Yaskawa INFORM job: UF_SELECTIE.JBI

/JOB
//NAME UF_SELECTIE
//POS
///NPOS 0,0,0,6,0,0
///USER 15
///TOOL 1
///POSTYPE USER
///RECTAN
///RCONF 1,0,0,0,0,0,0,0,0,0,0,0,0,0,0,0,0,0,0,0,0,0,0,0
P00100=0.001,-0.002,0.001,159.0512,-20.0126,15.9786
///USER 16
///RCONF 0,0,0,0,1,0,0,0,0,0,0,0,0,0,0,0,0,0,0,0,0,0,0,0
P00101=0.509,-0.968,-5.555,-18.4625,20.9980,-13.7043
///RCONF 1,0,0,0,0,0,0,0,0,0,0,0,0,0,0,0,0,0,0,0,0,0,0,0
P00120=-60.612,0.501,180.447,-18.4625,20.9980,-13.7043
P00121=0.001,-0.002,0.001,-18.4625,20.9980,-13.7043
///POSTYPE ROBOT
P00122=750.004,162.000,576.437,180.0000,-9.9968,0.0000
P00123=1150.002,160.000,520.003,180.0000,-25.0002,0.0000
//INST
///DATE 2025/05/06 14:51
///ATTR SC,RW
///GROUP1 RB1
///LVARS 0,10,20,0,0,0,0,0
NOP
SET B050 16
SET LI001 3
SET LI002 4
SET LI003 5
'
JUMP LABEL: B050
*15
FOR LI000 START= 120 TO 123
	 GETE LD[LI001] P[LI000] (1)
	 GETE LD[LI002] P[LI000] (2)
	 GETE LD[LI003] P[LI000] (3)
	 GETE LD000 P100 (4)
	 GETE LD001 P100 (5)
	 GETE LD002 P100 (6)
	 CNVRT PX[LI000] PX[LI000] UF#(15)
	 SETE P[LI000] (1) LD[LI001]
	 SETE P[LI000] (2) LD[LI002]
	 SETE P[LI000] (3) LD[LI003]
	 SETE P[LI000] (4) LD000
	 SETE P[LI000] (5) LD001
	 SETE P[LI000] (6) LD002
	 ADD LI001 3
	 ADD LI002 3
	 ADD LI003 3
NEXT LI000
JUMP *EINDE
'
*16
FOR LI000 START= 120 TO 123
	 GETE LD[LI001] P[LI000] (1)
	 GETE LD[LI002] P[LI000] (2)
	 GETE LD[LI003] P[LI000] (3)
	 GETE LD000 P101 (4)
	 GETE LD001 P101 (5)
	 GETE LD002 P101 (6)
	 CNVRT PX[LI000] PX[LI000] UF#(16)
	 SETE P[LI000] (1) LD[LI001]
	 SETE P[LI000] (2) LD[LI002]
	 MUL LD[LI002] -1
	 MUL LD[LI003] -1
	 SETE P[LI000] (3) LD[LI003]
	 SETE P[LI000] (4) LD000
	 SETE P[LI000] (5) LD001
	 SETE P[LI000] (6) LD002
	 ADD LI001 3
	 ADD LI002 3
	 ADD LI003 3
NEXT LI000
*EINDE
'P120
'
MOVJ P120 VJ=50.00
MOVL P121 V=250.0
ARCON
MOVL P122 V=4.2
ARCOF
MOVL P123 V=250.0
END
